ABB RobotStudio station: abb_linear_axis.rspag

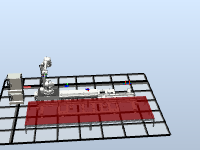
--- station ---
Station LinearAxis (saved by RobotStudio 6.7.7850.130)
Controller vController1, task T_ROB1: task frame (RAPID world) sits at (3503, -2050, 812) mm in the station
Controller vController1
  mechanical unit TRACK_1: IRBT2005_IRB_DBL1_INT_0_0_5__01, 1 joints, base frame (0, 0, 0) mm
  mechanical unit ROB_1: IRB4600_40_255_C_01_1, 6 joints, base frame (0, 0, 0) mm
Layout (positions relative to the parent item):
  - IRBT2005_IRB_DBL1_INT_0_0_5__01 [mechanism] at (2678.5, -2342, 352) mm; joint values [-1.9255] (rad or m)
      links: Base, Link1
  - IRB4600_40_255_C_01_1 [mechanism, from Robots\IRB4600_40_255_C_G_01.rslib] at (1577.5, -2050, 812) mm; joint values [-1.5708, 0, 0, 0, 0.4413, 0] (rad or m)
  - GenrerllCellEquipment  [graphiccomponentgroup, from Libraries\GenrerllCellEquipment .rslib]
    - MAS_Build_Platform [part, from Libraries\GenrerllCellEquipment .rslib] at (-3, 24.44, -100.55) mm
    - BachmannBase [part, from Libraries\GenrerllCellEquipment .rslib] at (0, 0, -100) mm
  - IRC5_Rob1 [graphiccomponentgroup]
    - IRC5_Drive-Module [part, from Libraries\IRC5_Drive-Module.rslib] at (-93.18, -1551.32, 0) mm, rotated rx 90 ry 0 rz 0 deg
    - IRC5_Singel-Cabinet [part, from Libraries\IRC5_Singel-Cabinet.rslib] at (-93.18, -1551.32, 646.49) mm, rotated rx 90 ry 0 rz 0 deg
  - ToolDummy [part] at (1577.5, -3617.06, 2519.34) mm, rotated rx -180 ry 64.71 rz 90 deg
Attachment: IRB4600_40_255_C_01_1 is attached to IRBT2005_IRB_DBL1_INT_0_0_5__01 / Link1
Attachment: IRC5_Singel-Cabinet is attached to IRC5_Drive-Module
Attachment: ToolDummy is attached to IRB4600_40_255_C_01_1 / Link6
Targets, tools, work objects and paths stored in the station and not in the controller backup, written as RAPID:
! task T_ROB1
MODULE Module1
  TASK PERS robtarget pPath_10:=[[2100.000441934,100.001285464,249.99750249],[-0.000000833,1,0.000000875,-0.000000188],[-1,0,1,0],[-1000,9E+09,9E+09,9E+09,9E+09,9E+09]];
  TASK PERS robtarget pPath_20:=[[1900.000680949,100.000196641,250.000172222],[0.000000147,1,0.000000374,0.000000054],[-1,0,1,0],[-1000,9E+09,9E+09,9E+09,9E+09,9E+09]];
  TASK PERS robtarget pHome:=[[-999.999655917,-1096.096640471,916.753202167],[0.24184468,0.664462964,0.664463172,-0.241844604],[-1,0,-1,0],[-1000,9E+09,9E+09,9E+09,9E+09,9E+09]];
ENDMODULE


--- Backups/vController1/RAPID/TASK1/PROGMOD/ROS_motion.mod ---
MODULE ROS_motion

! Software License Agreement (BSD License)
!
! Copyright (c) 2012, Edward Venator, Case Western Reserve University
! Copyright (c) 2012, Jeremy Zoss, Southwest Research Institute
! All rights reserved.
!
! Redistribution and use in source and binary forms, with or without modification,
! are permitted provided that the following conditions are met:
!
!   Redistributions of source code must retain the above copyright notice, this
!       list of conditions and the following disclaimer.
!   Redistributions in binary form must reproduce the above copyright notice, this
!       list of conditions and the following disclaimer in the documentation
!       and/or other materials provided with the distribution.
!   Neither the name of the Case Western Reserve University nor the names of its contributors
!       may be used to endorse or promote products derived from this software without
!       specific prior written permission.
!
! THIS SOFTWARE IS PROVIDED BY THE COPYRIGHT HOLDERS AND CONTRIBUTORS "AS IS" AND ANY
! EXPRESS OR IMPLIED WARRANTIES, INCLUDING, BUT NOT LIMITED TO, THE IMPLIED WARRANTIES
! OF MERCHANTABILITY AND FITNESS FOR A PARTICULAR PURPOSE ARE DISCLAIMED. IN NO EVENT
! SHALL THE COPYRIGHT HOLDER OR CONTRIBUTORS BE LIABLE FOR ANY DIRECT, INDIRECT,
! INCIDENTAL, SPECIAL, EXEMPLARY, OR CONSEQUENTIAL DAMAGES (INCLUDING, BUT NOT LIMITED
! TO, PROCUREMENT OF SUBSTITUTE GOODS OR SERVICES; LOSS OF USE, DATA, OR PROFITS; OR
! BUSINESS INTERRUPTION) HOWEVER CAUSED AND ON ANY THEORY OF LIABILITY, WHETHER IN
! CONTRACT, STRICT LIABILITY, OR TORT (INCLUDING NEGLIGENCE OR OTHERWISE) ARISING IN ANY
! WAY OUT OF THE USE OF THIS SOFTWARE, EVEN IF ADVISED OF THE POSSIBILITY OF SUCH DAMAGE.

LOCAL CONST zonedata DEFAULT_CORNER_DIST := z10;
LOCAL VAR ROS_joint_trajectory_pt trajectory{MAX_TRAJ_LENGTH};
LOCAL VAR num trajectory_size := 0;
LOCAL VAR intnum intr_new_trajectory;

PROC main()
    VAR num current_index;
    VAR jointtarget target;
    VAR speeddata move_speed := v10;  ! default speed
    VAR zonedata stop_mode;
    VAR bool skip_move;

    ! Set up interrupt to watch for new trajectory
    IDelete intr_new_trajectory;    ! clear interrupt handler, in case restarted with ExitCycle
    CONNECT intr_new_trajectory WITH new_trajectory_handler;
    IPers ROS_new_trajectory, intr_new_trajectory;

    WHILE true DO
        ! Check for new Trajectory
        IF (ROS_new_trajectory)
            init_trajectory;

        ! execute all points in this trajectory
        IF (trajectory_size > 0) THEN
            FOR current_index FROM 1 TO trajectory_size DO
                target.robax := trajectory{current_index}.joint_pos;
                target.extax := trajectory{current_index}.extax_pos;

                skip_move := (current_index = 1) AND is_near(target, 0.1, 0.1);

                stop_mode := DEFAULT_CORNER_DIST;  ! assume we're smoothing between points
                IF (current_index = trajectory_size) stop_mode := fine;  ! stop at path end

                ! Execute move command
                IF (NOT skip_move)
                    MoveAbsJ target, move_speed, \T:=trajectory{current_index}.duration, stop_mode, tool0;
            ENDFOR

            trajectory_size := 0;  ! trajectory done
        ENDIF

        WaitTime 0.05;  ! Throttle loop while waiting for new command
    ENDWHILE
ERROR
    ErrWrite \W, "Motion Error", "Error executing motion.  Aborting trajectory.";
    abort_trajectory;
ENDPROC

LOCAL PROC init_trajectory()
    clear_path;                    ! cancel any active motions

    WaitTestAndSet ROS_trajectory_lock;  ! acquire data-lock
      trajectory := ROS_trajectory;            ! copy to local var
      trajectory_size := ROS_trajectory_size;  ! copy to local var
      ROS_new_trajectory := FALSE;
    ROS_trajectory_lock := FALSE;         ! release data-lock
ENDPROC

LOCAL FUNC bool is_near(jointtarget target, num deg_tol, num mm_tol)
    VAR jointtarget curr_jnt;

    curr_jnt := CJointT();

    ! either an external axis is unconfigured/not present OR if it is, then it must be close enough
    RETURN ( ABS(curr_jnt.robax.rax_1 - target.robax.rax_1) < deg_tol )
       AND ( ABS(curr_jnt.robax.rax_2 - target.robax.rax_2) < deg_tol )
       AND ( ABS(curr_jnt.robax.rax_3 - target.robax.rax_3) < deg_tol )
       AND ( ABS(curr_jnt.robax.rax_4 - target.robax.rax_4) < deg_tol )
       AND ( ABS(curr_jnt.robax.rax_5 - target.robax.rax_5) < deg_tol )
       AND ( ABS(curr_jnt.robax.rax_6 - target.robax.rax_6) < deg_tol )
       AND ( (curr_jnt.extax.eax_a = 9E9) OR (ABS(curr_jnt.extax.eax_a - target.extax.eax_a) < mm_tol) )
       AND ( (curr_jnt.extax.eax_b = 9E9) OR (ABS(curr_jnt.extax.eax_b - target.extax.eax_b) < mm_tol) )
       AND ( (curr_jnt.extax.eax_c = 9E9) OR (ABS(curr_jnt.extax.eax_c - target.extax.eax_c) < mm_tol) )
       AND ( (curr_jnt.extax.eax_d = 9E9) OR (ABS(curr_jnt.extax.eax_d - target.extax.eax_d) < mm_tol) );
ENDFUNC

LOCAL PROC abort_trajectory()
    trajectory_size := 0;  ! "clear" local trajectory
    clear_path;
    ExitCycle;  ! restart program
ENDPROC

LOCAL PROC clear_path()
    IF ( NOT (IsStopMoveAct(\FromMoveTask) OR IsStopMoveAct(\FromNonMoveTask)) )
        StopMove;          ! stop any active motions
    ClearPath;             ! clear queued motion commands
    StartMove;             ! re-enable motions
ENDPROC

LOCAL TRAP new_trajectory_handler
    IF (NOT ROS_new_trajectory) RETURN;

    abort_trajectory;
ENDTRAP

ENDMODULE

--- Backups/vController1/RAPID/TASK1/SYSMOD/LINKEDM.sys ---
%%%
  VERSION:1
  LANGUAGE:ENGLISH
%%%

MODULE LINKEDM (SYSMODULE)

! FOLLOWER
!     Name of electronically linked follower axis used by operator at teach pendent.
      PERS string l_f_axis_name{5}       :=  ["",  "", "", "", ""];

!     Name of the mechanical unit for follower axis.
      PERS string l_f_mecunt_n{5}  :=  ["", "", "", "", ""];

!     Linked follower axis number in the mechanical unit (first axis in mech. unit is number 1).
      PERS num l_f_axis_no{5}      :=  [0,          0,   0,  0,  0];

! MASTER
!     Name of the mechanical unit for linked master axis.
      PERS string l_m_mecunt_n{5} :=  ["", "", "", "", ""];

!     Linked master axis number in the mechanical unit (first axis in mech. unit is number 1).
!     See axis number table in documentation for different master mechanical units.
      PERS num l_m_axis_no{5}     :=  [0,  0,  0,  0,  0];

! POSITION OFFSET
!     The increase of the allowed offset position between the master and follower
!     positions, used when starting AUTO mode. As soon as the offset is decreased
!     the old configurated parameter is used.
!     Example: 3 => the configurated value of allowed offset is increased 3 times.
      PERS num offset_ratio{5}       :=  [10,  10,   10,  10,  10];

! SPEED RATIO
!     Speed_ratio used in AUTO and JOG modes [ very_slow   slow    normal    fast]
!     Value 1 = max allowed manual speed.
      CONST num speed_ratio {20}      := [0.01, 0.01, 0.01, 0.01, 0.01,
                                          0.05, 0.05, 0.05, 0.05, 0.05,
                                          0.20, 0.20, 0.20, 0.20, 0.20,
                                          1.00, 1.00, 1.00, 1.00, 1.00];

! STEP SIZE
!     Displacement position used in JOG mode for each activation of positive or
!     negative movement.                  [very_short    short   normal   long]
!     Unit degees or meter.
      CONST num displacement {20}     := [0.001, 0.001, 0.001, 0.001, 0.001,
                                          0.005, 0.005, 0.005, 0.005, 0.005,
                                          0.020, 0.020, 0.020, 0.020, 0.020,
                                          0.100, 0.100, 0.100, 0.100, 0.100];


!-------------------------------------------------------------
 PROC Linked_m ()
      Linked_m_exe ;
 ENDPROC
ENDMODULE

--- Backups/vController1/RAPID/TASK1/SYSMOD/ROS_common.sys ---
MODULE ROS_common(SYSMODULE)

! Software License Agreement (BSD License)
!
! Copyright (c) 2012, Edward Venator, Case Western Reserve University
! Copyright (c) 2012, Jeremy Zoss, Southwest Research Institute
! All rights reserved.
!
! Redistribution and use in source and binary forms, with or without modification,
! are permitted provided that the following conditions are met:
!
!   Redistributions of source code must retain the above copyright notice, this
!       list of conditions and the following disclaimer.
!   Redistributions in binary form must reproduce the above copyright notice, this
!       list of conditions and the following disclaimer in the documentation
!       and/or other materials provided with the distribution.
!   Neither the name of the Case Western Reserve University nor the names of its contributors
!       may be used to endorse or promote products derived from this software without
!       specific prior written permission.
!
! THIS SOFTWARE IS PROVIDED BY THE COPYRIGHT HOLDERS AND CONTRIBUTORS "AS IS" AND ANY
! EXPRESS OR IMPLIED WARRANTIES, INCLUDING, BUT NOT LIMITED TO, THE IMPLIED WARRANTIES
! OF MERCHANTABILITY AND FITNESS FOR A PARTICULAR PURPOSE ARE DISCLAIMED. IN NO EVENT
! SHALL THE COPYRIGHT HOLDER OR CONTRIBUTORS BE LIABLE FOR ANY DIRECT, INDIRECT,
! INCIDENTAL, SPECIAL, EXEMPLARY, OR CONSEQUENTIAL DAMAGES (INCLUDING, BUT NOT LIMITED
! TO, PROCUREMENT OF SUBSTITUTE GOODS OR SERVICES; LOSS OF USE, DATA, OR PROFITS; OR
! BUSINESS INTERRUPTION) HOWEVER CAUSED AND ON ANY THEORY OF LIABILITY, WHETHER IN
! CONTRACT, STRICT LIABILITY, OR TORT (INCLUDING NEGLIGENCE OR OTHERWISE) ARISING IN ANY
! WAY OUT OF THE USE OF THIS SOFTWARE, EVEN IF ADVISED OF THE POSSIBILITY OF SUCH DAMAGE.

RECORD ROS_joint_trajectory_pt
	robjoint joint_pos;
    extjoint extax_pos;
	num duration;
ENDRECORD

CONST num MAX_TRAJ_LENGTH := 100;

! These variables should use TestAndSet read/write protection to prevent conflicts
PERS bool ROS_trajectory_lock := FALSE;
PERS ROS_joint_trajectory_pt ROS_trajectory{MAX_TRAJ_LENGTH};
PERS num ROS_trajectory_size := 0;
PERS bool ROS_new_trajectory := FALSE;       ! can safely READ, but should use lock to WRITE

ENDMODULE

--- Backups/vController1/RAPID/TASK1/SYSMOD/ROS_messages.sys ---
MODULE ROS_messages(SYSMODULE)
! Software License Agreement (BSD License)
!
! Copyright (c) 2012, Jeremy Zoss, Southwest Research Institute
! All rights reserved.
!
! Redistribution and use in source and binary forms, with or without modification,
! are permitted provided that the following conditions are met:
!
!   Redistributions of source code must retain the above copyright notice, this
!       list of conditions and the following disclaimer.
!   Redistributions in binary form must reproduce the above copyright notice, this
!       list of conditions and the following disclaimer in the documentation
!       and/or other materials provided with the distribution.
!   Neither the name of the Case Western Reserve University nor the names of its contributors
!       may be used to endorse or promote products derived from this software without
!       specific prior written permission.
!
! THIS SOFTWARE IS PROVIDED BY THE COPYRIGHT HOLDERS AND CONTRIBUTORS "AS IS" AND ANY
! EXPRESS OR IMPLIED WARRANTIES, INCLUDING, BUT NOT LIMITED TO, THE IMPLIED WARRANTIES
! OF MERCHANTABILITY AND FITNESS FOR A PARTICULAR PURPOSE ARE DISCLAIMED. IN NO EVENT
! SHALL THE COPYRIGHT HOLDER OR CONTRIBUTORS BE LIABLE FOR ANY DIRECT, INDIRECT,
! INCIDENTAL, SPECIAL, EXEMPLARY, OR CONSEQUENTIAL DAMAGES (INCLUDING, BUT NOT LIMITED
! TO, PROCUREMENT OF SUBSTITUTE GOODS OR SERVICES; LOSS OF USE, DATA, OR PROFITS; OR
! BUSINESS INTERRUPTION) HOWEVER CAUSED AND ON ANY THEORY OF LIABILITY, WHETHER IN
! CONTRACT, STRICT LIABILITY, OR TORT (INCLUDING NEGLIGENCE OR OTHERWISE) ARISING IN ANY
! WAY OUT OF THE USE OF THIS SOFTWARE, EVEN IF ADVISED OF THE POSSIBILITY OF SUCH DAMAGE.

RECORD ROS_msg_header
    num msg_type;
    num comm_type;
    num reply_code;
ENDRECORD

RECORD ROS_msg
    ROS_msg_header header;
    rawbytes data;
ENDRECORD

RECORD ROS_msg_joint_traj_pt
    ROS_msg_header header;
    num sequence_id;
    robjoint joints;  ! in DEGREES
    extjoint ext_axes;
    num velocity;
    num duration;
ENDRECORD

RECORD ROS_msg_joint_data
    ROS_msg_header header;
    num sequence_id;
    robjoint joints;  ! in DEGREES
    extjoint ext_axes;
ENDRECORD

! Message Type Codes (from simple_message/simple_message.h)
CONST num ROS_MSG_TYPE_INVALID       := 0;
CONST num ROS_MSG_TYPE_JOINT         := 10;  ! joint-position feedback
CONST num ROS_MSG_TYPE_JOINT_TRAJ_PT := 11;  ! joint-trajectory-point (for path downloading)
CONST num ROS_COM_TYPE_TOPIC         := 1;
CONST num ROS_COM_TYPE_SRV_REQ       := 2;
CONST num ROS_COM_TYPE_SRV_REPLY     := 3;
CONST num ROS_REPLY_TYPE_INVALID     := 0;
CONST num ROS_REPLY_TYPE_SUCCESS     := 1;
CONST num ROS_REPLY_TYPE_FAILURE     := 2;

! "Special" Sequence Codes (from simple_message/joint_traj_pt.h)
CONST num ROS_TRAJECTORY_START_DOWNLOAD := -1;
CONST num ROS_TRAJECTORY_END := -3;
CONST num ROS_TRAJECTORY_STOP := -4;

! Other message constants
CONST num ROS_MSG_MAX_JOINTS := 10;  ! from joint_data.h

PROC ROS_receive_msg_joint_traj_pt(VAR socketdev client_socket, VAR ROS_msg_joint_traj_pt message, \num wait_time)
    VAR ROS_msg raw_message;

    ! Read raw message data
    IF Present(wait_time) THEN
        ROS_receive_msg client_socket, raw_message, \wait_time:=wait_time;
    ELSE
        ROS_receive_msg client_socket, raw_message;
    ENDIF

    ! Integrity Check: Message Type
    IF (raw_message.header.msg_type <> ROS_MSG_TYPE_JOINT_TRAJ_PT) THEN
        ErrWrite \W, "ROS Socket Type Mismatch", "Unexpected message type",
                \RL2:="expected: " + ValToStr(ROS_MSG_TYPE_JOINT_TRAJ_PT),
                \RL3:="received: " + ValToStr(raw_message.header.msg_type);
        RAISE ERR_ARGVALERR;  ! TBD: define specific error code
    ENDIF

    ! Integrity Check: Data Size
    IF (RawBytesLen(raw_message.data) < 52) THEN
        ErrWrite \W, "ROS Socket Missing Data", "Insufficient data for joint_trajectory_pt",
                \RL2:="expected: 52",
                \RL3:="received: " + ValToStr(RawBytesLen(raw_message.data));
        RAISE ERR_OUTOFBND;  ! TBD: define specific error code
    ENDIF

    ! Copy Header data
    message.header := raw_message.header;

    ! Unpack data fields
    UnpackRawBytes raw_message.data, 1, message.sequence_id, \IntX:=DINT;
    UnpackRawBytes raw_message.data, 5, message.joints.rax_1, \Float4;
    UnpackRawBytes raw_message.data, 9, message.joints.rax_2, \Float4;
    UnpackRawBytes raw_message.data, 13, message.joints.rax_3, \Float4;
    UnpackRawBytes raw_message.data, 17, message.joints.rax_4, \Float4;
    UnpackRawBytes raw_message.data, 21, message.joints.rax_5, \Float4;
    UnpackRawBytes raw_message.data, 25, message.joints.rax_6, \Float4;
    UnpackRawBytes raw_message.data, 29, message.ext_axes.eax_a, \Float4;
    UnpackRawBytes raw_message.data, 33, message.ext_axes.eax_b, \Float4;
    UnpackRawBytes raw_message.data, 37, message.ext_axes.eax_c, \Float4;
    UnpackRawBytes raw_message.data, 41, message.ext_axes.eax_d, \Float4;
    UnpackRawBytes raw_message.data, 45, message.velocity, \Float4;
    UnpackRawBytes raw_message.data, 49, message.duration, \Float4;

    ! Convert data from ROS units to ABB units
    message.joints := rad2deg_robjoint(message.joints);
    message.ext_axes := m2mm_extjoint(message.ext_axes);
    ! TBD: convert velocity

ERROR
    RAISE;  ! raise errors to calling code
ENDPROC

PROC ROS_send_msg_joint_data(VAR socketdev client_socket, ROS_msg_joint_data message)
    VAR ROS_msg raw_message;
    VAR robjoint ROS_joints;
    VAR extjoint ROS_ext_axes;
    VAR num i;

    ! Force message header to the correct values
    raw_message.header.msg_type := ROS_MSG_TYPE_JOINT;
    raw_message.header.comm_type := ROS_COM_TYPE_TOPIC;
    raw_message.header.reply_code := ROS_REPLY_TYPE_INVALID;

    ! Convert data from ABB units to ROS units
    ROS_joints := deg2rad_robjoint(message.joints);
    ROS_ext_axes := mm2m_extjoint(message.ext_axes);

    ! Pack data into message
    PackRawBytes message.sequence_id, raw_message.data,  1, \IntX:=DINT;
    PackRawBytes ROS_joints.rax_1,    raw_message.data,  5, \Float4;
    PackRawBytes ROS_joints.rax_2,    raw_message.data,  9, \Float4;
    PackRawBytes ROS_joints.rax_3,    raw_message.data, 13, \Float4;
    PackRawBytes ROS_joints.rax_4,    raw_message.data, 17, \Float4;
    PackRawBytes ROS_joints.rax_5,    raw_message.data, 21, \Float4;
    PackRawBytes ROS_joints.rax_6,    raw_message.data, 25, \Float4;
    PackRawBytes ROS_ext_axes.eax_a,  raw_message.data, 29, \Float4;
    PackRawBytes ROS_ext_axes.eax_b,  raw_message.data, 33, \Float4;
    PackRawBytes ROS_ext_axes.eax_c,  raw_message.data, 37, \Float4;
    PackRawBytes ROS_ext_axes.eax_d,  raw_message.data, 41, \Float4;

    ROS_send_msg client_socket, raw_message;

ERROR
    RAISE;  ! raise errors to calling code
ENDPROC

LOCAL FUNC num deg2rad(num deg)
    RETURN deg * pi / 180;
ENDFUNC

LOCAL FUNC num connected_eax(num eax)
    ! The value 9E9 is defined for axes which are not connected
    IF eax <> 9E9 THEN
        RETURN eax;
    ENDIF
    RETURN 0;
ENDFUNC

! Returns only connected external axes in METERS
LOCAL FUNC extjoint mm2m_extjoint(extjoint all_eax)
    VAR extjoint eax;
    eax.eax_a := connected_eax(all_eax.eax_a) / 1000;
    eax.eax_b := connected_eax(all_eax.eax_b) / 1000;
    eax.eax_c := connected_eax(all_eax.eax_c) / 1000;
    eax.eax_d := connected_eax(all_eax.eax_d) / 1000;
    RETURN eax;
ENDFUNC

! Returns external axes in MILLIMETERS
LOCAL FUNC extjoint m2mm_extjoint(extjoint eax_in_m)
    VAR extjoint eax_in_mm;
    eax_in_mm.eax_a := eax_in_m.eax_a * 1000;
    eax_in_mm.eax_b := eax_in_m.eax_b * 1000;
    eax_in_mm.eax_c := eax_in_m.eax_c * 1000;
    eax_in_mm.eax_d := eax_in_m.eax_d * 1000;

    RETURN eax_in_mm;
ENDFUNC

LOCAL FUNC robjoint deg2rad_robjoint(robjoint deg)
    VAR robjoint rad;
    rad.rax_1 := deg2rad(deg.rax_1);
    rad.rax_2 := deg2rad(deg.rax_2);
    rad.rax_3 := deg2rad(deg.rax_3);
    rad.rax_4 := deg2rad(deg.rax_4);
    rad.rax_5 := deg2rad(deg.rax_5);
    rad.rax_6 := deg2rad(deg.rax_6);

    RETURN rad;
ENDFUNC

LOCAL FUNC num rad2deg(num rad)
    RETURN rad * 180 / pi;
ENDFUNC

LOCAL FUNC robjoint rad2deg_robjoint(robjoint rad)
    VAR robjoint deg;
    deg.rax_1 := rad2deg(rad.rax_1);
    deg.rax_2 := rad2deg(rad.rax_2);
    deg.rax_3 := rad2deg(rad.rax_3);
    deg.rax_4 := rad2deg(rad.rax_4);
    deg.rax_5 := rad2deg(rad.rax_5);
    deg.rax_6 := rad2deg(rad.rax_6);

    RETURN deg;
ENDFUNC

ENDMODULE

--- Backups/vController1/RAPID/TASK1/SYSMOD/ROS_socket.sys ---
MODULE ROS_socket(SYSMODULE)
! Software License Agreement (BSD License)
!
! Copyright (c) 2012, Jeremy Zoss, Southwest Research Institute
! Copyright (c) 2012, Edward Venator, Case Western Reserve University
! All rights reserved.
!
! Redistribution and use in source and binary forms, with or without modification,
! are permitted provided that the following conditions are met:
!
!   Redistributions of source code must retain the above copyright notice, this
!       list of conditions and the following disclaimer.
!   Redistributions in binary form must reproduce the above copyright notice, this
!       list of conditions and the following disclaimer in the documentation
!       and/or other materials provided with the distribution.
!   Neither the name of the Case Western Reserve University nor the names of its contributors
!       may be used to endorse or promote products derived from this software without
!       specific prior written permission.
!
! THIS SOFTWARE IS PROVIDED BY THE COPYRIGHT HOLDERS AND CONTRIBUTORS "AS IS" AND ANY
! EXPRESS OR IMPLIED WARRANTIES, INCLUDING, BUT NOT LIMITED TO, THE IMPLIED WARRANTIES
! OF MERCHANTABILITY AND FITNESS FOR A PARTICULAR PURPOSE ARE DISCLAIMED. IN NO EVENT
! SHALL THE COPYRIGHT HOLDER OR CONTRIBUTORS BE LIABLE FOR ANY DIRECT, INDIRECT,
! INCIDENTAL, SPECIAL, EXEMPLARY, OR CONSEQUENTIAL DAMAGES (INCLUDING, BUT NOT LIMITED
! TO, PROCUREMENT OF SUBSTITUTE GOODS OR SERVICES; LOSS OF USE, DATA, OR PROFITS; OR
! BUSINESS INTERRUPTION) HOWEVER CAUSED AND ON ANY THEORY OF LIABILITY, WHETHER IN
! CONTRACT, STRICT LIABILITY, OR TORT (INCLUDING NEGLIGENCE OR OTHERWISE) ARISING IN ANY
! WAY OUT OF THE USE OF THIS SOFTWARE, EVEN IF ADVISED OF THE POSSIBILITY OF SUCH DAMAGE.

PROC ROS_init_socket(VAR socketdev server_socket, num port)
    IF (SocketGetStatus(server_socket) = SOCKET_CLOSED) SocketCreate server_socket;
    IF (SocketGetStatus(server_socket) = SOCKET_CREATED) SocketBind server_socket, "0.0.0.0", port;
    IF (SocketGetStatus(server_socket) = SOCKET_BOUND) SocketListen server_socket;

ERROR
    RAISE;  ! raise errors to calling code
ENDPROC

PROC ROS_wait_for_client(VAR socketdev server_socket, VAR socketdev client_socket, \num wait_time)
    VAR string client_ip;
    VAR num time_val := WAIT_MAX;  ! default to wait-forever

    IF Present(wait_time) time_val := wait_time;

    IF (SocketGetStatus(client_socket) <> SOCKET_CLOSED) SocketClose client_socket;
    WaitUntil (SocketGetStatus(client_socket) = SOCKET_CLOSED);

    SocketAccept server_socket, client_socket, \ClientAddress:=client_ip, \Time:=time_val;
    TPWrite "Client at "+client_ip+" connected.";

ERROR
    RAISE;  ! raise errors to calling code
ENDPROC

PROC ROS_receive_msg(VAR socketdev client_socket, VAR ROS_msg message, \num wait_time)
    VAR rawbytes buffer;
    VAR num time_val := WAIT_MAX;  ! default to wait-forever
    VAR num bytes_rcvd;
    VAR num msg_length;

    ClearRawBytes buffer;
    IF Present(wait_time) time_val := wait_time;

    ! TBD: need to determine whether this handles split/merged messages correctly

    ! Read prefix INT (total message length)
    SocketReceive client_socket, \RawData:=buffer, \ReadNoOfBytes:=4, \Time:=time_val;
    UnpackRawBytes buffer, 1, msg_length, \IntX:=UDINT;

    ! Read remaining message bytes
    SocketReceive client_socket, \RawData:=buffer, \ReadNoOfBytes:=msg_length, \NoRecBytes:=bytes_rcvd, \Time:=time_val;
    IF (bytes_rcvd <> msg_length) THEN
        ErrWrite \W, "ROS Socket Recv Failed", "Did not receive expected # of bytes.",
                 \RL2:="Expected: " + ValToStr(msg_length),
                 \RL3:="Received: " + ValToStr(bytes_rcvd);
        RETURN;
    ENDIF

    ! Unpack message header/data
    UnpackRawBytes buffer, 1, message.header.msg_type, \IntX:=DINT;
    UnpackRawBytes buffer, 5, message.header.comm_type, \IntX:=DINT;
    UnpackRawBytes buffer, 9, message.header.reply_code, \IntX:=DINT;
    CopyRawBytes   buffer, 13, message.data, 1;

ERROR
    RAISE;  ! raise errors to calling code
ENDPROC

PROC ROS_send_msg(VAR socketdev client_socket, VAR ROS_msg message)
    VAR rawbytes buffer;

    PackRawBytes 12 + RawBytesLen(message.data), buffer,  1, \IntX := UDINT; ! Packet length (excluding this prefix)
    PackRawBytes message.header.msg_type,        buffer,  5, \IntX := DINT;  ! Message type
    PackRawBytes message.header.comm_type,       buffer,  9, \IntX := DINT;  ! Comm type
    PackRawBytes message.header.reply_code,      buffer, 13, \IntX := DINT;  ! Reply code
    CopyRawBytes message.data, 1,                buffer, 17;                 ! Message data

    SocketSend client_socket \RawData:=buffer;

ERROR
    RAISE;  ! raise errors to calling code
ENDPROC

ENDMODULE

--- Backups/vController1/RAPID/TASK3/PROGMOD/ROS_stateServer.mod ---
MODULE ROS_stateServer

! Software License Agreement (BSD License)
!
! Copyright (c) 2012, Edward Venator, Case Western Reserve University
! Copyright (c) 2012, Jeremy Zoss, Southwest Research Institute
! All rights reserved.
!
! Redistribution and use in source and binary forms, with or without modification,
! are permitted provided that the following conditions are met:
!
!   Redistributions of source code must retain the above copyright notice, this
!       list of conditions and the following disclaimer.
!   Redistributions in binary form must reproduce the above copyright notice, this
!       list of conditions and the following disclaimer in the documentation
!       and/or other materials provided with the distribution.
!   Neither the name of the Case Western Reserve University nor the names of its contributors
!       may be used to endorse or promote products derived from this software without
!       specific prior written permission.
!
! THIS SOFTWARE IS PROVIDED BY THE COPYRIGHT HOLDERS AND CONTRIBUTORS "AS IS" AND ANY
! EXPRESS OR IMPLIED WARRANTIES, INCLUDING, BUT NOT LIMITED TO, THE IMPLIED WARRANTIES
! OF MERCHANTABILITY AND FITNESS FOR A PARTICULAR PURPOSE ARE DISCLAIMED. IN NO EVENT
! SHALL THE COPYRIGHT HOLDER OR CONTRIBUTORS BE LIABLE FOR ANY DIRECT, INDIRECT,
! INCIDENTAL, SPECIAL, EXEMPLARY, OR CONSEQUENTIAL DAMAGES (INCLUDING, BUT NOT LIMITED
! TO, PROCUREMENT OF SUBSTITUTE GOODS OR SERVICES; LOSS OF USE, DATA, OR PROFITS; OR
! BUSINESS INTERRUPTION) HOWEVER CAUSED AND ON ANY THEORY OF LIABILITY, WHETHER IN
! CONTRACT, STRICT LIABILITY, OR TORT (INCLUDING NEGLIGENCE OR OTHERWISE) ARISING IN ANY
! WAY OUT OF THE USE OF THIS SOFTWARE, EVEN IF ADVISED OF THE POSSIBILITY OF SUCH DAMAGE.

LOCAL CONST num server_port := 11002;
LOCAL CONST num update_rate := 0.10;  ! broadcast rate (sec)

LOCAL VAR socketdev server_socket;
LOCAL VAR socketdev client_socket;

PROC main()

    TPWrite "StateServer: Waiting for connection.";
	ROS_init_socket server_socket, server_port;
    ROS_wait_for_client server_socket, client_socket;

	WHILE (TRUE) DO
		send_joints;
		WaitTime update_rate;
    ENDWHILE

ERROR (ERR_SOCK_TIMEOUT, ERR_SOCK_CLOSED)
	IF (ERRNO=ERR_SOCK_TIMEOUT) OR (ERRNO=ERR_SOCK_CLOSED) THEN
        SkipWarn;  ! TBD: include this error data in the message logged below?
        ErrWrite \W, "ROS StateServer disconnect", "Connection lost.  Waiting for new connection.";
        ExitCycle;  ! restart program
	ELSE
		TRYNEXT;
	ENDIF
UNDO
ENDPROC

LOCAL PROC send_joints()
	VAR ROS_msg_joint_data message;
	VAR jointtarget joints;

    ! get current joint position (degrees)
	joints := CJointT();

    ! create message
    message.header := [ROS_MSG_TYPE_JOINT, ROS_COM_TYPE_TOPIC, ROS_REPLY_TYPE_INVALID];
    message.sequence_id := 0;
    message.joints := joints.robax;
    message.ext_axes := joints.extax;

    ! send message to client
    ROS_send_msg_joint_data client_socket, message;

ERROR
    RAISE;  ! raise errors to calling code
ENDPROC

ENDMODULE

--- Backups/vController1/RAPID/TASK4/PROGMOD/ROS_motionServer.mod ---
MODULE ROS_motionServer

! Software License Agreement (BSD License)
!
! Copyright (c) 2012, Edward Venator, Case Western Reserve University
! Copyright (c) 2012, Jeremy Zoss, Southwest Research Institute
! All rights reserved.
!
! Redistribution and use in source and binary forms, with or without modification,
! are permitted provided that the following conditions are met:
!
!   Redistributions of source code must retain the above copyright notice, this
!       list of conditions and the following disclaimer.
!   Redistributions in binary form must reproduce the above copyright notice, this
!       list of conditions and the following disclaimer in the documentation
!       and/or other materials provided with the distribution.
!   Neither the name of the Case Western Reserve University nor the names of its contributors
!       may be used to endorse or promote products derived from this software without
!       specific prior written permission.
!
! THIS SOFTWARE IS PROVIDED BY THE COPYRIGHT HOLDERS AND CONTRIBUTORS "AS IS" AND ANY
! EXPRESS OR IMPLIED WARRANTIES, INCLUDING, BUT NOT LIMITED TO, THE IMPLIED WARRANTIES
! OF MERCHANTABILITY AND FITNESS FOR A PARTICULAR PURPOSE ARE DISCLAIMED. IN NO EVENT
! SHALL THE COPYRIGHT HOLDER OR CONTRIBUTORS BE LIABLE FOR ANY DIRECT, INDIRECT,
! INCIDENTAL, SPECIAL, EXEMPLARY, OR CONSEQUENTIAL DAMAGES (INCLUDING, BUT NOT LIMITED
! TO, PROCUREMENT OF SUBSTITUTE GOODS OR SERVICES; LOSS OF USE, DATA, OR PROFITS; OR
! BUSINESS INTERRUPTION) HOWEVER CAUSED AND ON ANY THEORY OF LIABILITY, WHETHER IN
! CONTRACT, STRICT LIABILITY, OR TORT (INCLUDING NEGLIGENCE OR OTHERWISE) ARISING IN ANY
! WAY OUT OF THE USE OF THIS SOFTWARE, EVEN IF ADVISED OF THE POSSIBILITY OF SUCH DAMAGE.

LOCAL CONST num server_port := 11000;

LOCAL VAR socketdev server_socket;
LOCAL VAR socketdev client_socket;
LOCAL VAR ROS_joint_trajectory_pt trajectory{MAX_TRAJ_LENGTH};
LOCAL VAR num trajectory_size;

PROC main()
    VAR ROS_msg_joint_traj_pt message;

    TPWrite "MotionServer: Waiting for connection.";
	ROS_init_socket server_socket, server_port;
    ROS_wait_for_client server_socket, client_socket;

    WHILE ( true ) DO
		! Recieve Joint Trajectory Pt Message
        ROS_receive_msg_joint_traj_pt client_socket, message;
		trajectory_pt_callback message;
	ENDWHILE

ERROR (ERR_SOCK_TIMEOUT, ERR_SOCK_CLOSED)
	IF (ERRNO=ERR_SOCK_TIMEOUT) OR (ERRNO=ERR_SOCK_CLOSED) THEN
        SkipWarn;  ! TBD: include this error data in the message logged below?
        ErrWrite \W, "ROS MotionServer disconnect", "Connection lost.  Resetting socket.";
		ExitCycle;  ! restart program
	ELSE
		TRYNEXT;
	ENDIF
UNDO
	IF (SocketGetStatus(client_socket) <> SOCKET_CLOSED) SocketClose client_socket;
	IF (SocketGetStatus(server_socket) <> SOCKET_CLOSED) SocketClose server_socket;
ENDPROC

LOCAL PROC trajectory_pt_callback(ROS_msg_joint_traj_pt message)
	VAR ROS_joint_trajectory_pt point;
	VAR jointtarget current_pos;
    VAR ROS_msg reply_msg;

    point := [message.joints, message.ext_axes, message.duration];

    ! use sequence_id to signal start/end of trajectory download
	TEST message.sequence_id
		CASE ROS_TRAJECTORY_START_DOWNLOAD:
            TPWrite "Traj START received";
			trajectory_size := 0;                 ! Reset trajectory size
            add_traj_pt point;                    ! Add this point to the trajectory
		CASE ROS_TRAJECTORY_END:
            TPWrite "Traj END received";
            add_traj_pt point;                    ! Add this point to the trajectory
            activate_trajectory;
		CASE ROS_TRAJECTORY_STOP:
            TPWrite "Traj STOP received";
            trajectory_size := 0;  ! empty trajectory
            activate_trajectory;
            StopMove; ClearPath; StartMove;  ! redundant, but re-issue stop command just to be safe
		DEFAULT:
            add_traj_pt point;                    ! Add this point to the trajectory
	ENDTEST

    ! send reply, if requested
    IF (message.header.comm_type = ROS_COM_TYPE_SRV_REQ) THEN
        reply_msg.header := [ROS_MSG_TYPE_JOINT_TRAJ_PT, ROS_COM_TYPE_SRV_REPLY, ROS_REPLY_TYPE_SUCCESS];
        ROS_send_msg client_socket, reply_msg;
    ENDIF

ERROR
    RAISE;  ! raise errors to calling code
ENDPROC

LOCAL PROC add_traj_pt(ROS_joint_trajectory_pt point)
    IF (trajectory_size = MAX_TRAJ_LENGTH) THEN
        ErrWrite \W, "Too Many Trajectory Points", "Trajectory has already reached its maximum size",
            \RL2:="max_size = " + ValToStr(MAX_TRAJ_LENGTH);
    ELSE
        Incr trajectory_size;
        trajectory{trajectory_size} := point; !Add this point to the trajectory
    ENDIF
ENDPROC

LOCAL PROC activate_trajectory()
    WaitTestAndSet ROS_trajectory_lock;  ! acquire data-lock
    TPWrite "Sending " + ValToStr(trajectory_size) + " points to MOTION task";
    ROS_trajectory := trajectory;
    ROS_trajectory_size := trajectory_size;
    ROS_new_trajectory := TRUE;
    ROS_trajectory_lock := FALSE;  ! release data-lock
ENDPROC

ENDMODULE

--- Backups/vController1/SYSPAR/EIO.cfg ---
EIO:CFG_1.0:6:1::
#
INDUSTRIAL_NETWORK:

      -Name "DeviceNet" -Label "DeviceNet Master/Slave Network" -Address "2"

      -Name "PROFINET" -Connection "PROFINET Network"\
      -Label "PROFINET Controller/Device Network"\
      -CfgPath "160725_A005_MAS1_ProfinetKonfig_PF.xml" -StationName "Master1"
#
DEVICENET_INTERNAL_DEVICE:

      -Name "DN_Internal_Device" -VendorName "ABB Robotics"\
      -ProductName "DeviceNet Internal Slave Device"
#
PROFINET_INTERNAL_DEVICE:

      -Name "PN_Internal_Device" -VendorName "ABB Robotics"\
      -ProductName "PROFINET Internal Device"
#
PROFINET_DEVICE:

      -Name "Unit1" -StationName "EK9300"
#
EIO_SIGNAL:

      -Name "diGr1Scan" -SignalType "DI" -Device "Unit1"\
      -Label "Unit 1 Sick light sensor" -DeviceMap "0" -Access "All"

      -Name "diGr1Res2" -SignalType "DI" -Device "Unit1"\
      -Label "Unit 1 Digital Input Reserve" -DeviceMap "1" -Access "All"

      -Name "diGr1Res3" -SignalType "DI" -Device "Unit1"\
      -Label "Unit 1 Digital Input Reserve" -DeviceMap "2" -Access "All"

      -Name "diGr1Res4" -SignalType "DI" -Device "Unit1"\
      -Label "Unit 1 Digital Input Reserve" -DeviceMap "3" -Access "All"

      -Name "diGr1Res5" -SignalType "DI" -Device "Unit1"\
      -Label "Unit 1 Digital Input Reserve" -DeviceMap "4" -Access "All"

      -Name "diGr1Res6" -SignalType "DI" -Device "Unit1"\
      -Label "Unit 1 Digital Input Reserve" -DeviceMap "5" -Access "All"

      -Name "diGr1Res7" -SignalType "DI" -Device "Unit1"\
      -Label "Unit 1 Digital Input Reserve" -DeviceMap "6" -Access "All"

      -Name "diGr1Res8" -SignalType "DI" -Device "Unit1"\
      -Label "Unit 1 Digital Input Reserve" -DeviceMap "7" -Access "All"

      -Name "doGr1NailGun1On" -SignalType "DO" -Device "Unit1"\
      -Label "Unit 1 Nailgun 1 On" -DeviceMap "0" -Access "All"

      -Name "doGr1NailGun2On" -SignalType "DO" -Device "Unit1"\
      -Label "Unit 1 Nailgun 2 On" -DeviceMap "1" -Access "All"

      -Name "doGr1VacuumOn" -SignalType "DO" -Device "Unit1"\
      -Label "Unit 1 Vacuum On" -DeviceMap "2" -Access "All"

      -Name "doGr1Res4" -SignalType "DO" -Device "Unit1"\
      -Label "Unit 1 Digital Output Reserve" -DeviceMap "3" -Access "All"

      -Name "doGr1Res5" -SignalType "DO" -Device "Unit1"\
      -Label "Unit 1 Digital Output Reserve" -DeviceMap "4" -Access "All"

      -Name "doGr1Res6" -SignalType "DO" -Device "Unit1"\
      -Label "Unit 1 Digital Output Reserve" -DeviceMap "5" -Access "All"

      -Name "doGr1Res7" -SignalType "DO" -Device "Unit1"\
      -Label "Unit 1 Digital Output Reserve" -DeviceMap "6" -Access "All"

      -Name "doGr1Res8" -SignalType "DO" -Device "Unit1"\
      -Label "Unit 1 Digital Output Reserve" -DeviceMap "7" -Access "All"

      -Name "voNewPart" -SignalType "DO"
